{attribute addProperty BoxType "EPP1518-0002-0016"}
{attribute addProperty Id "StatusAT %I*Status_DA5A5D41162"}
{attribute addProperty CRC "696262572"}
{attribute addProperty SizeInBites "16"}
{attribute addProperty SizeInBytes "2"}
TYPE DIG_Inputs_Device_29801FAC :
STRUCT
	{attribute addProperty Name "Status"}
	Status AT %I* : Status_DA5A5D41;
END_STRUCT
END_TYPE

(* stored: Version 1.2.0.0, ProductVersion 3.1.4024.9
   DUT DIG_Inputs_Device_29801FAC: Id {bc046503-4920-4e20-8456-c18ea38dbabb} *)
